// TwinCAT 3 PLC project TcoLoggers
// Title: TcoLoggers
// Company: Vortex.Library
// ProjectVersion: 0.4.2.535
// ProgramVersion: 3.1.4023.0
// libraries:
//   Tc2_Standard, * (Beckhoff Automation GmbH)
//   Tc2_System, * (Beckhoff Automation GmbH)
//   Tc2_Utilities, * (Beckhoff Automation GmbH)
//   Tc3_JsonXml, * (Beckhoff Automation GmbH)
//   Tc3_Module, * (Beckhoff Automation GmbH)
//   TcoCore, 0.4.2.535 (Vortex.Library)
// project tree:
//   / PlcTask.TcTTO
//   POUs/TcoLoggers/Enrichers/ InstancePathEnricher.TcPOU
//   POUs/TcoLoggers/ ITcoArguments.TcIO (not stored), ITcoLogEnricher.TcIO (not stored), ITcoLogger.TcIO, ITcoLogSink.TcIO (not stored), LogEnricherList.TcPOU (not stored), LogEvent.TcDUT (not stored), LogLevel.TcDUT, LogSinkList.TcPOU, TcoArguments.TcPOU (not stored), TcoLogger.TcPOU (not stored), TcoLoggerConfiguration.TcPOU, TcoLoggerEnrichmentConfiguration.TcPOU, TcoLoggerSinkConfiguration.TcPOU
//   POUs/TcoLoggers/Sinks/ AdsLogSink.TcPOU (not stored), VolatileSink.TcPOU (not stored)
//   POUs/TcoLoggers/UserExtensions/ ExtendedLoggerEnrichmentConfiguration.TcPOU, ExtendedLoggerSinkConfiguration.TcPOU (not stored), FileSink.TcPOU, ProjectNameEnricher.TcPOU
//   POUs/ MAIN.TcPOU
// real-time tasks:
//   TASK PlcTask: cycle T#10ms, priority 20, ADS port 350
//   TASK PlcTask1: cycle T#10ms, priority 21, ADS port 351

CONFIGURATION TcoLoggers
    RESOURCE PLC ON TwinCAT3
        TASK PlcTask(INTERVAL := T#10ms, PRIORITY := 20);
        PROGRAM MAIN WITH PlcTask : MAIN;
    END_RESOURCE
END_CONFIGURATION

// ---- POUs/TcoLoggers/LogLevel.TcDUT
{attribute 'qualified_only'}
{attribute 'strict'}
TYPE LogLevel :
(
	Debug := 0,
	Info,
	Warning,
	Error,
	Fatal
);
END_TYPE

// ---- POUs/TcoLoggers/ITcoLogger.TcIO
//TODO
INTERFACE ITcoLogger

(*~
		<docu>
			<summary>
				Adds message of 'debug' category to the message queue.				 
			</summary>		
		</docu>
~*)
METHOD PUBLIC Debug
VAR_INPUT
	(*~
		<docu>
			<summary>
				Arbitrary message string.			 
			</summary>			
		</docu>
	~*)
	Message : STRING(255);
END_VAR
END_METHOD

(*~
		<docu>
			<summary>
				Adds message of 'error' category to the message queue.				 
			</summary>						
		</docu>
~*)
METHOD PUBLIC Error
VAR_INPUT
	(*~
		<docu>
			<summary>
				Arbitrary message string.			 
			</summary>			
		</docu>
	~*)
	Message : STRING(255);
END_VAR
END_METHOD

(*~
		<docu>
			<summary>
				Adds message of 'critical' category to the message queue.				 
			</summary>						
		</docu>
~*)
METHOD PUBLIC Fatal
VAR_INPUT
	(*~
		<docu>
			<summary>
				Arbitrary message string.			 
			</summary>			
		</docu>
	~*)
	Message : STRING(255);
END_VAR
END_METHOD

METHOD ForContext : ITcoLogger
VAR_INPUT
	Context		: ITcoContext;
END_VAR
END_METHOD

METHOD ForIdentity : ITcoLogger
VAR_INPUT
	Identity	: ULINT;
END_VAR
END_METHOD

(*~
		<docu>
			<summary>
				Adds message of 'information' category to the message queue.				 
			</summary>			
		</docu>
~*)
METHOD PUBLIC Info 
VAR_INPUT
	(*~
		<docu>
			<summary>
				Arbitrary message string.			 
			</summary>			
		</docu>
	~*)
	Message : STRING(255);
END_VAR
END_METHOD

(*~
		<docu>
			<summary>
				Adds message of 'warning' category to the message queue.				 
			</summary>					
		</docu>
~*)
METHOD PUBLIC Warning 
VAR_INPUT
	(*~
		<docu>
			<summary>
				Arbitrary message string.			 
			</summary>			
		</docu>
	~*)
	Message : STRING(255);
END_VAR
END_METHOD

METHOD WithArgs : ITcoArguments
VAR_INPUT
END_VAR
END_METHOD

END_INTERFACE

// ---- POUs/MAIN.TcPOU
PROGRAM MAIN
VAR
   
END_VAR

END_PROGRAM

// ---- POUs/TcoLoggers/Enrichers/InstancePathEnricher.TcPOU
{attribute 'reflection'}
FUNCTION_BLOCK FINAL InstancePathEnricher IMPLEMENTS ITcoLogEnricher
VAR_INPUT
END_VAR
VAR_OUTPUT
END_VAR
VAR
	{attribute 'instance-path'} 
    {attribute 'noinit'} 
    _instancePath : STRING(255); 
END_VAR

METHOD Enrich : BOOL
VAR_INPUT
	LogEvent	: REFERENCE TO LogEvent;
END_VAR

VAR
	info		: STRING;
END_VAR
IF NOT __ISVALIDREF(LogEvent) THEN
	RETURN;
END_IF

info := CONCAT('[', _instancePath);
info := CONCAT(info, '] ');

// e.g. [MAIN.Infeed.Conveyor] My log message
LogEvent.Text := CONCAT(info, LogEvent.Text);
END_METHOD

END_FUNCTION_BLOCK

// ---- POUs/TcoLoggers/LogSinkList.TcPOU
FUNCTION_BLOCK LogSinkList
VAR_INPUT
END_VAR
VAR_OUTPUT
END_VAR
VAR
	_count		: UINT;
	_iterator			: UINT;
	//~
	_sinks				: ARRAY[0..(MAX_SINKS - 1)] OF ITcoLogSink;
	//~
END_VAR

VAR CONSTANT
	MAX_SINKS				: USINT := 10;
END_VAR

METHOD PUBLIC AddSink : BOOL
VAR_INPUT
	Sink	: ITcoLogSink;
END_VAR
IF _count >= MAX_SINKS - 1 THEN
	AddSink := FALSE;
	RETURN;
END_IF

IF Sink = NULL THEN
	AddSink := FALSE;
	RETURN;
END_IF

_count := _count + 1;
_sinks[_count] := Sink;

AddSink := TRUE;
END_METHOD

METHOD PUBLIC Clear : BOOL
VAR
	i : DINT;
END_VAR
FOR i := 1 TO (MAX_SINKS - 1) DO
	_sinks[i] := NULL;
END_FOR

_count	:= 0;
_iterator		:= 0;
END_METHOD

PROPERTY PUBLIC Count : UINT
GET
Count := _count;
END_GET
END_PROPERTY

METHOD PUBLIC GetNext : ITcoLogSink
VAR_INPUT
END_VAR
_iterator := _iterator + 1;
GetNext := _sinks[_iterator];
END_METHOD

METHOD PUBLIC HasNext : BOOL
VAR_INPUT
END_VAR
IF _iterator < _count THEN
	HasNext := TRUE;
	RETURN;
END_IF

HasNext := FALSE;
END_METHOD

PROPERTY PUBLIC IsEmpty : BOOL
GET
IsEmpty := _count = 0;
END_GET
END_PROPERTY

METHOD PUBLIC ResetIterator : BOOL
VAR_INPUT
END_VAR
_iterator := 0;
END_METHOD

END_FUNCTION_BLOCK

// ---- POUs/TcoLoggers/TcoLoggerConfiguration.TcPOU
FUNCTION_BLOCK TcoLoggerConfiguration
VAR_INPUT
END_VAR
VAR_OUTPUT
END_VAR
VAR
	_minimumLevel			: LogLevel := LogLevel.Info;
	
	_sinks					: LogSinkList;
	_enrichers				: LogEnricherList;

	_enrichmentConfig		: TcoLoggerEnrichmentConfiguration := ( Config := THIS^);
	_sinksConfig			: TcoLoggerSinkConfiguration := ( Config := THIS^);
END_VAR

METHOD INTERNAL AddEnrichment : BOOL
VAR_INPUT
	Enricher		: ITcoLogEnricher;
END_VAR
AddEnrichment := _enrichers.AddEnricher(Enricher);
END_METHOD

METHOD INTERNAL AddSink : BOOL
VAR_INPUT
	Sink		: ITcoLogSink;
END_VAR
AddSink := _sinks.AddSink(Sink);
END_METHOD

METHOD PUBLIC Build : BOOL
VAR_INPUT
END_VAR
Build := TRUE;
END_METHOD

METHOD PUBLIC Clear : REFERENCE TO TcoLoggerConfiguration
VAR_INPUT
END_VAR
_minimumLevel := LogLevel.Info;

_sinks.Clear();
MEMSET(ADR(_enrichers), 0, SIZEOF(_enrichers));

Clear REF= THIS^;
END_METHOD

PROPERTY INTERNAL Enrichers : REFERENCE TO LogEnricherList
GET
Enrichers REF= _enrichers;
END_GET
END_PROPERTY

PROPERTY EnrichWith : REFERENCE TO TcoLoggerEnrichmentConfiguration
GET
EnrichWith REF= _enrichmentConfig;
END_GET
END_PROPERTY

PROPERTY PUBLIC Level : LogLevel
GET
Level := _minimumLevel;
END_GET
END_PROPERTY

METHOD PUBLIC MinimumLevel : REFERENCE TO TcoLoggerConfiguration
VAR_INPUT
	Level		: LogLevel;
END_VAR
_minimumLevel := Level;
MinimumLevel REF= THIS^;
END_METHOD

METHOD PUBLIC ReadFrom : REFERENCE TO TcoLoggerConfiguration
VAR_INPUT
	FilePath		: STRING(255);
END_VAR
// Read json config file

// json structure example

(*
{
    "MinimumLevel": "Debug",
    "WriteTo": [
      { "Name": "XAE" },
      { "Name": "File", "Args": { "path": "C:/Temp/log.txt" } }
    ],
    "Enrich": [ "Context", "InstancePath", "ProjectName" ]
}
*)

ReadFrom REF= THIS^;
END_METHOD

PROPERTY INTERNAL Sinks : REFERENCE TO LogSinkList
GET
Sinks REF= _sinks;
END_GET
END_PROPERTY

PROPERTY PUBLIC WriteTo : REFERENCE TO TcoLoggerSinkConfiguration
GET
WriteTo REF= _sinksConfig;
END_GET
END_PROPERTY

END_FUNCTION_BLOCK

// ---- POUs/TcoLoggers/TcoLoggerEnrichmentConfiguration.TcPOU
FUNCTION_BLOCK TcoLoggerEnrichmentConfiguration

VAR_INPUT
	Config		: REFERENCE TO TcoLoggerConfiguration;
END_VAR

VAR
	_instancePathEnricher 	: InstancePathEnricher;
END_VAR

METHOD PUBLIC Context : REFERENCE TO TcoLoggerConfiguration
VAR_INPUT
END_VAR
Context REF= Config;
END_METHOD

METHOD PUBLIC CycleCount : REFERENCE TO TcoLoggerConfiguration
VAR_INPUT
END_VAR
CycleCount REF= Config;
END_METHOD

METHOD PUBLIC InstancePath : REFERENCE TO TcoLoggerConfiguration
VAR_INPUT
END_VAR
Config.AddEnrichment(_instancePathEnricher);
InstancePath REF= Config;
END_METHOD

END_FUNCTION_BLOCK

// ---- POUs/TcoLoggers/TcoLoggerSinkConfiguration.TcPOU
FUNCTION_BLOCK TcoLoggerSinkConfiguration 

VAR_INPUT
	Config		: REFERENCE TO TcoLoggerConfiguration;
END_VAR

VAR
	_xaeSink		: AdsLogSink;
	_volatileSink	: VolatileSink;
END_VAR

METHOD PUBLIC Memory : REFERENCE TO TcoLoggerConfiguration
VAR_INPUT
END_VAR
Config.AddSink(_volatileSink);
Memory REF= Config;
END_METHOD

METHOD PUBLIC XAE : REFERENCE TO TcoLoggerConfiguration
VAR_INPUT
END_VAR
Config.AddSink(_xaeSink);
XAE := Config;
END_METHOD

END_FUNCTION_BLOCK

// ---- POUs/TcoLoggers/UserExtensions/ExtendedLoggerEnrichmentConfiguration.TcPOU
FUNCTION_BLOCK FINAL ExtendedLoggerEnrichmentConfiguration EXTENDS TcoLoggerEnrichmentConfiguration
VAR_INPUT
END_VAR
VAR_OUTPUT
END_VAR
VAR
	_projectNameEnricher		: ProjectNameEnricher;
END_VAR

METHOD PUBLIC ProjectName : REFERENCE TO TcoLoggerConfiguration
VAR_INPUT
END_VAR
_config.AddEnrichment(_projectNameEnricher);
ProjectName := _config;
END_METHOD

END_FUNCTION_BLOCK

// ---- POUs/TcoLoggers/UserExtensions/ProjectNameEnricher.TcPOU
FUNCTION_BLOCK FINAL ProjectNameEnricher IMPLEMENTS ITcoLogEnricher
VAR_INPUT
END_VAR
VAR_OUTPUT
END_VAR
VAR
END_VAR

METHOD Enrich : BOOL
VAR_INPUT
	LogEvent	: REFERENCE TO LogEvent;
END_VAR

VAR
	info		: STRING;
END_VAR
IF NOT __ISVALIDREF(LogEvent) THEN
	RETURN;
END_IF

info := CONCAT('[', _AppInfo.ProjectName);
info := CONCAT(info, '] ');

// e.g. [MyProjectName] My log message
LogEvent.Text := CONCAT(info, LogEvent.Text);
END_METHOD

END_FUNCTION_BLOCK

// ---- POUs/TcoLoggers/UserExtensions/FileSink.TcPOU
FUNCTION_BLOCK FileSink IMPLEMENTS ITcoLogSink
VAR_INPUT
END_VAR
VAR_OUTPUT
END_VAR
VAR
	_filePath		: STRING(255);
END_VAR

METHOD Emit : BOOL
VAR_INPUT
	LogEvent	: REFERENCE TO LogEvent;
END_VAR
// Write to file writer buffer


// e.g. use sample of benhar-dev
// https://github.com/benhar-dev/tc3-data-logger
END_METHOD

PROPERTY PUBLIC FilePath : STRING(255)
GET
FilePath := _filePath;
END_GET
SET
_filePath := FilePath;
END_SET
END_PROPERTY

END_FUNCTION_BLOCK
